PROGRAM POU
VAR
	dtVar : DATE_AND_TIME := DT#2023-02-07-13:10:00;
	pDateTime : POINTER TO DATE_AND_TIME;
END_VAR

pDateTime := ADR(dtVar);
pDateTime^ := DT#2023-02-08-15:31:19;

END_PROGRAM

(* stored: Version 1.1.0.1, ProductVersion 3.1.4024.12
   POU POU: Id {692759e6-f0e8-427c-9ada-964c908ff5a8}, SpecialFunc None *)
